PROGRAM MAIN
VAR
    _tcoIrc5TestContext : TcoSimpleTestContext;

    _wpfContext : WpfContext;
    _wpfContextCall : BOOL := FALSE;

END_VAR

_tcoIrc5TestContext.ProbeRun();


IF _wpfContextCall THEN
	_wpfContext.Run();
END_IF

END_PROGRAM

(* stored: Version 1.1.0.1, ProductVersion 3.1.4024.12
   POU MAIN: Id {20e36e6a-1247-05bf-1677-012e31b12f3e}, SpecialFunc None *)
